FUNCTION_BLOCK WAGOConveyorControllerParamatised (* Composite Function Block Type *)
  (* Standard: 61499-2 *)
  (* Version 0.2, 2003-12-05, JHC, Rockwell Automation, Renamed from NEWCOMPFB. *)
  (* Compiler header: package fb.rt.wago; *)
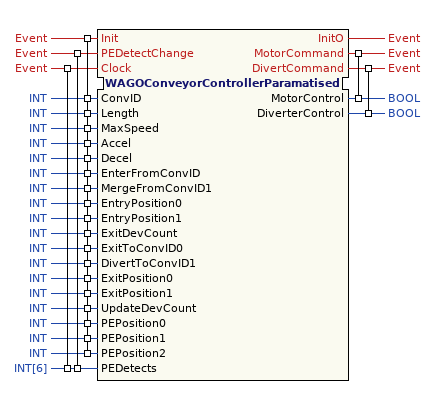
  EVENT_INPUT
    Init WITH ConvID, Length, MaxSpeed, EntryPosition0, EntryPosition1, ExitDevCount, ExitPosition0, ExitPosition1, UpdateDevCount, PEPosition0, PEPosition1, PEPosition2, EnterFromConvID, MergeFromConvID1, ExitToConvID0, DivertToConvID1, Accel, Decel; (* Initialization Request *)
    PEDetectChange WITH PEDetects; (* Instance of Time *)
    Clock WITH PEDetects;
  END_EVENT
  EVENT_OUTPUT
    InitO; (* Initialization Confirm *)
    MotorCommand WITH MotorControl;
    DivertCommand WITH DiverterControl;
  END_EVENT
  VAR_INPUT
    ConvID : INT; (* Input event qualifier *)
    Length : INT;
    MaxSpeed : INT;
    Accel : INT;
    Decel : INT;
    EnterFromConvID : INT; (* Input event qualifier *)
    MergeFromConvID1 : INT; (* Input event qualifier *)
    EntryPosition0 : INT; (* Input event qualifier *)
    EntryPosition1 : INT; (* Input event qualifier *)
    ExitDevCount : INT; (* Input event qualifier *)
    ExitToConvID0 : INT; (* Input event qualifier *)
    DivertToConvID1 : INT; (* Input event qualifier *)
    ExitPosition0 : INT; (* Input event qualifier *)
    ExitPosition1 : INT; (* Input event qualifier *)
    UpdateDevCount : INT; (* Input event qualifier *)
    PEPosition0 : INT; (* Input event qualifier *)
    PEPosition1 : INT; (* Input event qualifier *)
    PEPosition2 : INT; (* Input event qualifier *)
    PEDetects : ARRAY [0..5] OF INT; (* Input event qualifier *)
  END_VAR
  VAR_OUTPUT
    MotorControl : BOOL; (* true = go, false = stop *)
    DiverterControl : BOOL; (* true = Divert, false = DontDivert *)
  END_VAR
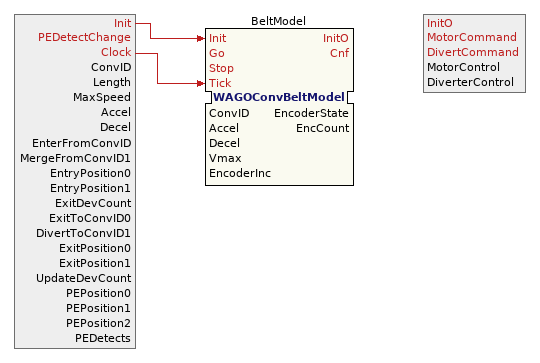
  FBS
    BeltModel : WAGOConvBeltModel;
  END_FBS
  EVENT_CONNECTIONS
    Init TO BeltModel.Init;
    Clock TO BeltModel.Tick;
  END_CONNECTIONS
END_FUNCTION_BLOCK
